Yaskawa INFORM job: TESTSRXG.JBI

/JOB
//NAME TESTSRXG
//POS
///NPOS 5,5,0,0,0,0
///TOOL 0
///POSTYPE PULSE
///PULSE
C00000=-135757,70063,29136,218,102808,36551
C00001=-135757,68735,33777,215,99269,36544
C00002=-135757,68588,34641,215,98660,36544
C00003=-135757,68558,34832,215,98527,36544
C00004=-132196,66266,32151,43,98993,37735
BC00000=182506,671659,131057
BC00001=182506,671659,131057
BC00002=182506,671659,131057
BC00003=182506,671659,131057
BC00004=182506,671659,131057
//INST
///DATE 2024/05/22 11:02
///ATTR SC,RW
///GROUP1 RB1,BS1
NOP
MOVJ C00000 BC00000 VJ=0.78
MOVL C00001 BC00001 V=11.0
REFP 1 C00002 BC00002
CALL JOB:SEARCH-R1-S13D
MOVL C00003 BC00003 V=11.0
REFP 1 C00004 BC00004
END
